TYPE TcoUrRobotics_O2T_Reg1_IO : 
STRUCT
    bArray AT %Q* : ARRAY[0..99] OF BYTE;
END_STRUCT
END_TYPE

(* stored: Version 1.1.0.1, ProductVersion 3.1.4024.12
   DUT TcoUrRobotics_O2T_Reg1_IO: Id {7f0c1e3e-daca-0faf-1d74-e03d83e126a1} *)
